{attribute addProperty BoxType "EL7041-0001-0016"}
{attribute addProperty Id "StatusAT %I*Status_B999DC12162"}
{attribute addProperty CRC "2172400331"}
{attribute addProperty SizeInBites "16"}
{attribute addProperty SizeInBytes "2"}
TYPE STM_Status_817C32CB :
STRUCT
	{attribute addProperty Name "Status"}
	Status AT %I* : Status_B999DC12;
END_STRUCT
END_TYPE

(* stored: Version 1.2.0.0, ProductVersion 3.1.4024.9
   DUT STM_Status_817C32CB: Id {9fe210a5-d30d-495a-99fa-28cbc234a199} *)
